VISUALIZATION STN400HMI  // 2x2
END_VISUALIZATION

(* stored: Version 1.1.0.1, ProductVersion 3.1.4024.2
   Visu STN400HMI: Id {9acb7116-0525-4bed-8ecd-5802c5b0eb8c} *)
